// TIA Portal V17 export
// export: Created 2025-05-06T13:48:20.4992801Z, ExportSetting WithDefaults, DisplayName Totally Integrated Automation Portal, DisplayVersion V17 Update 8, DisplayName TIA Portal Openness, DisplayVersion V17 Update 8, DisplayName TIA Portal Version Control Interface, DisplayVersion V17, DisplayName SINAMICS Startdrive Advanced, DisplayVersion V17 SP2, DisplayName SINAMICS Startdrive G110M, G120, G120C, G120D, G120P, G115D, DisplayVersion V17 SP2, DisplayName SINAMICS Startdrive G130, G150, S120, S150, SINAMICS MV, S210, DisplayVersion V17 SP2, DisplayName STEP 7 Professional, DisplayVersion V17 Update 8, DisplayName SINUMERIK ONE STEP 7 Toolbox, DisplayVersion V17 Update 12, DisplayName SINUMERIK 840D sl STEP 7 Toolbox, DisplayVersion V17 Update 12, DisplayName STEP 7 Safety, DisplayVersion V17 Update 6, DisplayName WinCC Advanced, DisplayVersion V17 Update 8
FUNCTION_BLOCK "FB2107_LIGHTS"   // FB2107, LAD
{ S7_Optimized_Access := 'TRUE' }
VERSION : 0.1
// stored: AutoNumber false, IsIECCheckEnabled false, IsRetainMemResEnabled false, MemoryReserve 100, SetENOAutomatically false, UDAEnableTagReadback false
   VAR_INPUT
      GENERAL_MACHINE_LIGHT_OPTION : Bool;
      CIRCUIT_BRAKER_IN : Bool;
      LIGHT_ON_SELECTOR : Bool;
      MANUAL_REQ_LINE : Bool;   // MANUAL REQUEST HMI LINE NUMBER
      SWITCH_ON_AUTO_REQ : Bool;   // SWITCH ON AUTO REQUEST
      SWITCH_OFF_AUTO_REQ : Bool;   // SWITCH OFF AUTO REQUEST
   END_VAR
   VAR_OUTPUT
      LIGHTS_ON : Bool;   // LIGHTS ON OUTPUT
      HMI_LINE_ON_EXEC : Bool;   // HMI LINE ON EXECUTABILITY
      HMI_LINE_OFF_EXEC : Bool;   // HMI LINE OFF EXECUTABILITY
      HMI_LINE_ON_STATUS : Bool;   // HMI LINE ON STATUS
      HMI_LINE_OFF_STATUS : Bool;   // HMI LINE OFF STATUS
   END_VAR
   VAR
      SWITCH_ON_GENERAL_CONDITIONS : Bool;   // SWITCH ON GENERAL CONDITIONS
      SWITCH_ON_INITIAL_CONDITIONS : Bool;   // SWITCH ON INITIAL CONDITIONS
      SWITCH_ON_MANUAL_REQ : Bool;   // SWITCH ON MANUAL REQUEST
      SWITCH_ON_GLOBAL_REQ : Bool;   // SWITCH ON GLOBAL REQUEST
      SWITCH_ON_COMMAND : Bool;   // SWITCH ON COMMAND
      SWITCH_ON : Bool;   // SWITCH ON
      IN_SERVICE : Bool;   // IN SERVICE
      SWITCH_OFF_GENERAL_CONDITIONS : Bool;   // SWITCH OFF GENERAL CONDITIONS
      SWITCH_OFF_INITIAL_CONDITIONS : Bool;   // SWITCH OFF INITIAL CONDITIONS
      SWITCH_OFF_MANUAL_REQ : Bool;   // SWITCH OFF MANUAL REQUEST
      SWITCH_OFF_GLOBAL_REQ : Bool;   // SWITCH OFF GLOBAL REQUEST
      SWITCH_OFF_COMMAND : Bool;   // SWITCH OFF COMMAND
      SWITCH_OFF : Bool;   // SWITCH OFF
      OUT_OF_SERVICE : Bool;   // OUT OF SERVICE
      SWITCH_ON_GLOBAL_REQUEST_AUX0 : Bool;   // SWITCH ON GLOBAL REQUEST AUXILIARY 0
      SWITCH_ON_GLOBAL_REQUEST_AUX1 : Bool;   // SWITCH ON GLOBAL REQUEST AUXILIARY 1
      SWITCH_ON_GLOBAL_REQUEST_AUX2 : Bool;   // SWITCH ON GLOBAL REQUEST AUXILIARY 2
      SWITCH_ON_GLOBAL_REQUEST_AUX3 : Bool;   // SWITCH ON GLOBAL REQUEST AUXILIARY 3
      SWITCH_OFF_GLOBAL_REQUEST_AUX1 : Bool;   // SWITCH OFF GLOBAL REQUEST AUXILIARY 1
      SWITCH_OFF_GLOBAL_REQUEST_AUX2 : Bool;   // SWITCH OFF GLOBAL REQUEST AUXILIARY 2
      SWITCH_OFF_DOORS_CLOSED_TIMER : IEC_TIMER;
      SWITCH_OFF_IN_SERVICE_DELAY_TIMER : IEC_TIMER;
   END_VAR
   // SWITCH_OFF_DOORS_CLOSED_TIMER.PT := T#10M;
   // SWITCH_OFF_IN_SERVICE_DELAY_TIMER.PT := T#1H;
   VAR_TEMP   // added for the SCL form of the ladder/FBD networks
      _w1 : Bool;
      _w2 : Bool;
      _w3 : Bool;
      _w4 : Bool;
      _w5 : Bool;
      _w6 : Bool;
   END_VAR
BEGIN

REGION Network 1: SWITCH ON GENERAL CONDITIONS
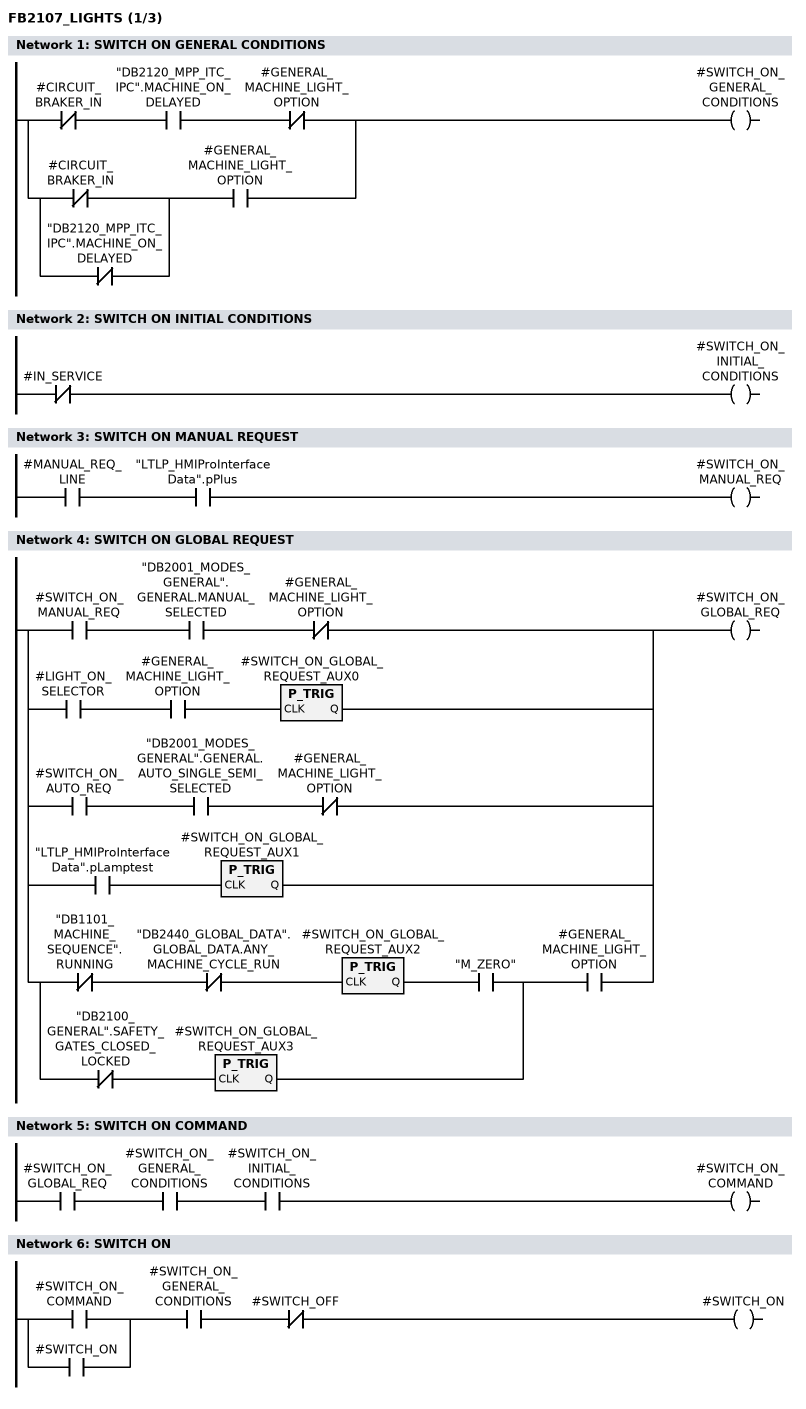
   RUNG wire#powerrail
      I_Contact( #CIRCUIT_BRAKER_IN )
      Contact( "DB2120_MPP_ITC_IPC".MACHINE_ON_DELAYED )
      I_Contact( #GENERAL_MACHINE_LIGHT_OPTION )
      wire#w1
      Coil( #SWITCH_ON_GENERAL_CONDITIONS )
   END_RUNG
   RUNG wire#powerrail
      I_Contact( #CIRCUIT_BRAKER_IN )
      wire#w2
      Contact( #GENERAL_MACHINE_LIGHT_OPTION )
   END_RUNG wire#w1
   RUNG wire#powerrail
      I_Contact( "DB2120_MPP_ITC_IPC".MACHINE_ON_DELAYED )
   END_RUNG wire#w2
   // the same network as SCL:
   #SWITCH_ON_GENERAL_CONDITIONS := (NOT #CIRCUIT_BRAKER_IN AND "DB2120_MPP_ITC_IPC".MACHINE_ON_DELAYED AND NOT #GENERAL_MACHINE_LIGHT_OPTION) OR ((NOT #CIRCUIT_BRAKER_IN OR NOT "DB2120_MPP_ITC_IPC".MACHINE_ON_DELAYED) AND #GENERAL_MACHINE_LIGHT_OPTION);
END_REGION

REGION Network 2: SWITCH ON INITIAL CONDITIONS
   RUNG wire#powerrail
      I_Contact( #IN_SERVICE )
      Coil( #SWITCH_ON_INITIAL_CONDITIONS )
   END_RUNG
   // the same network as SCL:
   #SWITCH_ON_INITIAL_CONDITIONS := NOT #IN_SERVICE;
END_REGION

REGION Network 3: SWITCH ON MANUAL REQUEST
   RUNG wire#powerrail
      Contact( #MANUAL_REQ_LINE )
      Contact( "LTLP_HMIProInterfaceData".pPlus )
      Coil( #SWITCH_ON_MANUAL_REQ )
   END_RUNG
   // the same network as SCL:
   #SWITCH_ON_MANUAL_REQ := #MANUAL_REQ_LINE AND "LTLP_HMIProInterfaceData".pPlus;
END_REGION

REGION Network 4: SWITCH ON GLOBAL REQUEST
   RUNG wire#powerrail
      Contact( #SWITCH_ON_MANUAL_REQ )
      Contact( "DB2001_MODES_GENERAL".GENERAL.MANUAL_SELECTED )
      I_Contact( #GENERAL_MACHINE_LIGHT_OPTION )
      wire#w1
      Coil( #SWITCH_ON_GLOBAL_REQ )
   END_RUNG
   RUNG wire#powerrail
      Contact( #LIGHT_ON_SELECTOR )
      Contact( #GENERAL_MACHINE_LIGHT_OPTION )
      P_Trig( #SWITCH_ON_GLOBAL_REQUEST_AUX0 )
   END_RUNG wire#w1
   RUNG wire#powerrail
      Contact( #SWITCH_ON_AUTO_REQ )
      Contact( "DB2001_MODES_GENERAL".GENERAL.AUTO_SINGLE_SEMI_SELECTED )
      I_Contact( #GENERAL_MACHINE_LIGHT_OPTION )
   END_RUNG wire#w1
   RUNG wire#powerrail
      Contact( "LTLP_HMIProInterfaceData".pLamptest )
      P_Trig( #SWITCH_ON_GLOBAL_REQUEST_AUX1 )
   END_RUNG wire#w1
   RUNG wire#powerrail
      I_Contact( "DB1101_MACHINE_SEQUENCE".RUNNING )
      I_Contact( "DB2440_GLOBAL_DATA".GLOBAL_DATA.ANY_MACHINE_CYCLE_RUN )
      P_Trig( #SWITCH_ON_GLOBAL_REQUEST_AUX2 )
      Contact( "M_ZERO" )
      wire#w2
      Contact( #GENERAL_MACHINE_LIGHT_OPTION )
   END_RUNG wire#w1
   RUNG wire#powerrail
      I_Contact( "DB2100_GENERAL".SAFETY_GATES_CLOSED_LOCKED )
      P_Trig( #SWITCH_ON_GLOBAL_REQUEST_AUX3 )
   END_RUNG wire#w2
   // the same network as SCL:
   #_w1 := #LIGHT_ON_SELECTOR AND #GENERAL_MACHINE_LIGHT_OPTION;
   #_w2 := #_w1 AND NOT #SWITCH_ON_GLOBAL_REQUEST_AUX0;   // rising edge
   #SWITCH_ON_GLOBAL_REQUEST_AUX0 := #_w1;
   #_w3 := "LTLP_HMIProInterfaceData".pLamptest AND NOT #SWITCH_ON_GLOBAL_REQUEST_AUX1;   // rising edge
   #SWITCH_ON_GLOBAL_REQUEST_AUX1 := "LTLP_HMIProInterfaceData".pLamptest;
   #_w4 := NOT "DB1101_MACHINE_SEQUENCE".RUNNING AND NOT "DB2440_GLOBAL_DATA".GLOBAL_DATA.ANY_MACHINE_CYCLE_RUN;
   #_w5 := #_w4 AND NOT #SWITCH_ON_GLOBAL_REQUEST_AUX2;   // rising edge
   #SWITCH_ON_GLOBAL_REQUEST_AUX2 := #_w4;
   #_w6 := NOT "DB2100_GENERAL".SAFETY_GATES_CLOSED_LOCKED AND NOT #SWITCH_ON_GLOBAL_REQUEST_AUX3;   // rising edge
   #SWITCH_ON_GLOBAL_REQUEST_AUX3 := NOT "DB2100_GENERAL".SAFETY_GATES_CLOSED_LOCKED;
   #SWITCH_ON_GLOBAL_REQ := (#SWITCH_ON_MANUAL_REQ AND "DB2001_MODES_GENERAL".GENERAL.MANUAL_SELECTED AND NOT #GENERAL_MACHINE_LIGHT_OPTION) OR #_w2 OR (#SWITCH_ON_AUTO_REQ AND "DB2001_MODES_GENERAL".GENERAL.AUTO_SINGLE_SEMI_SELECTED AND NOT #GENERAL_MACHINE_LIGHT_OPTION) OR #_w3 OR (((#_w5 AND "M_ZERO") OR #_w6) AND #GENERAL_MACHINE_LIGHT_OPTION);
END_REGION

REGION Network 5: SWITCH ON COMMAND
   RUNG wire#powerrail
      Contact( #SWITCH_ON_GLOBAL_REQ )
      Contact( #SWITCH_ON_GENERAL_CONDITIONS )
      Contact( #SWITCH_ON_INITIAL_CONDITIONS )
      Coil( #SWITCH_ON_COMMAND )
   END_RUNG
   // the same network as SCL:
   #SWITCH_ON_COMMAND := #SWITCH_ON_GLOBAL_REQ AND #SWITCH_ON_GENERAL_CONDITIONS AND #SWITCH_ON_INITIAL_CONDITIONS;
END_REGION

REGION Network 6: SWITCH ON
   RUNG wire#powerrail
      Contact( #SWITCH_ON_COMMAND )
      wire#w1
      Contact( #SWITCH_ON_GENERAL_CONDITIONS )
      I_Contact( #SWITCH_OFF )
      Coil( #SWITCH_ON )
   END_RUNG
   RUNG wire#powerrail
      Contact( #SWITCH_ON )
   END_RUNG wire#w1
   // the same network as SCL:
   #SWITCH_ON := (#SWITCH_ON_COMMAND OR #SWITCH_ON) AND #SWITCH_ON_GENERAL_CONDITIONS AND NOT #SWITCH_OFF;
END_REGION

REGION Network 7: IN SERVICE
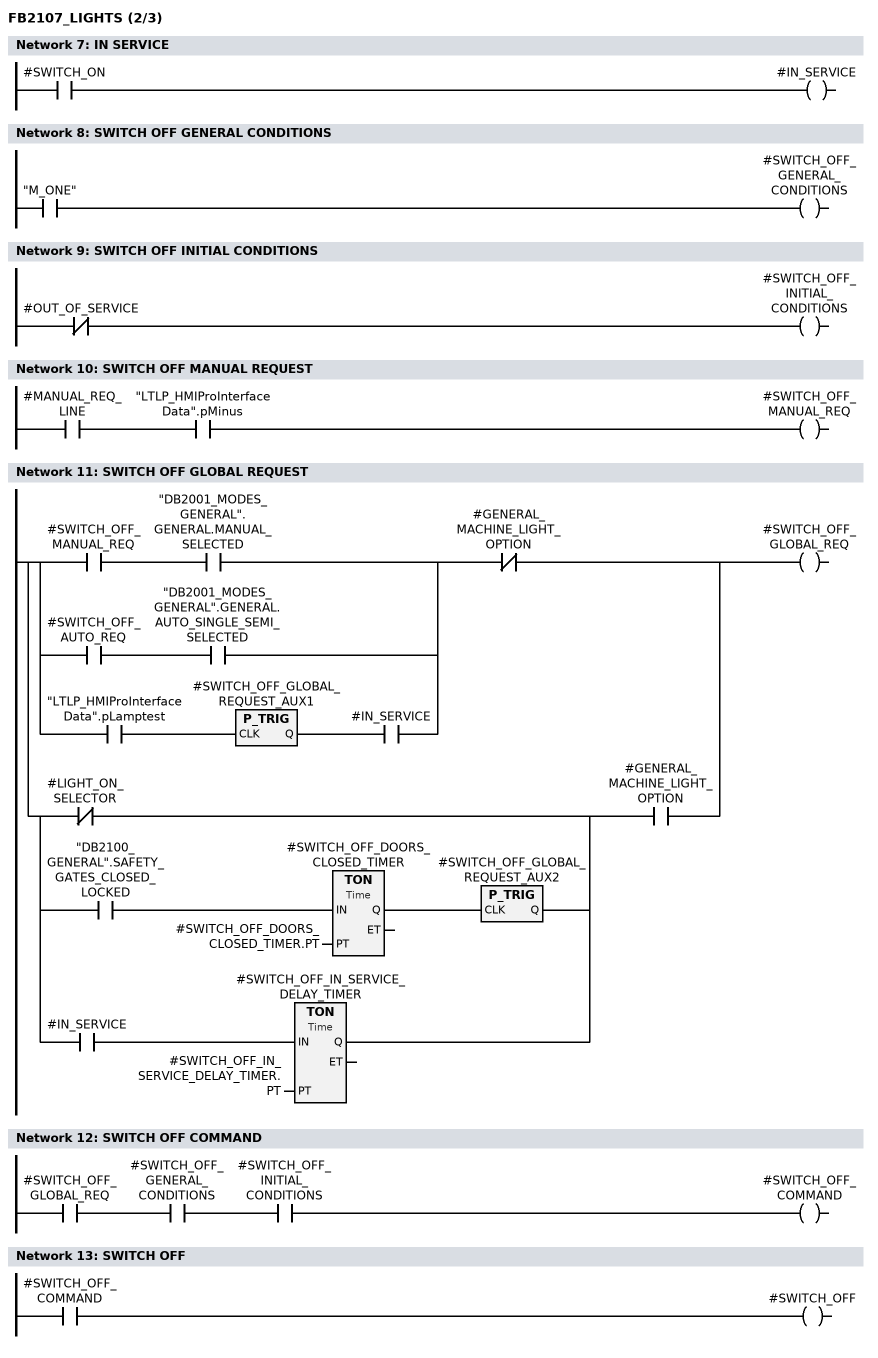
   RUNG wire#powerrail
      Contact( #SWITCH_ON )
      Coil( #IN_SERVICE )
   END_RUNG
   // the same network as SCL:
   #IN_SERVICE := #SWITCH_ON;
END_REGION

REGION Network 8: SWITCH OFF GENERAL CONDITIONS
   RUNG wire#powerrail
      Contact( "M_ONE" )
      Coil( #SWITCH_OFF_GENERAL_CONDITIONS )
   END_RUNG
   // the same network as SCL:
   #SWITCH_OFF_GENERAL_CONDITIONS := "M_ONE";
END_REGION

REGION Network 9: SWITCH OFF INITIAL CONDITIONS
   RUNG wire#powerrail
      I_Contact( #OUT_OF_SERVICE )
      Coil( #SWITCH_OFF_INITIAL_CONDITIONS )
   END_RUNG
   // the same network as SCL:
   #SWITCH_OFF_INITIAL_CONDITIONS := NOT #OUT_OF_SERVICE;
END_REGION

REGION Network 10: SWITCH OFF MANUAL REQUEST
   RUNG wire#powerrail
      Contact( #MANUAL_REQ_LINE )
      Contact( "LTLP_HMIProInterfaceData".pMinus )
      Coil( #SWITCH_OFF_MANUAL_REQ )
   END_RUNG
   // the same network as SCL:
   #SWITCH_OFF_MANUAL_REQ := #MANUAL_REQ_LINE AND "LTLP_HMIProInterfaceData".pMinus;
END_REGION

REGION Network 11: SWITCH OFF GLOBAL REQUEST
   RUNG wire#powerrail
      Contact( #SWITCH_OFF_MANUAL_REQ )
      Contact( "DB2001_MODES_GENERAL".GENERAL.MANUAL_SELECTED )
      wire#w1
      I_Contact( #GENERAL_MACHINE_LIGHT_OPTION )
      wire#w2
      Coil( #SWITCH_OFF_GLOBAL_REQ )
   END_RUNG
   RUNG wire#powerrail
      Contact( #SWITCH_OFF_AUTO_REQ )
      Contact( "DB2001_MODES_GENERAL".GENERAL.AUTO_SINGLE_SEMI_SELECTED )
   END_RUNG wire#w1
   RUNG wire#powerrail
      Contact( "LTLP_HMIProInterfaceData".pLamptest )
      P_Trig( #SWITCH_OFF_GLOBAL_REQUEST_AUX1 )
      Contact( #IN_SERVICE )
   END_RUNG wire#w1
   RUNG wire#powerrail
      I_Contact( #LIGHT_ON_SELECTOR )
      wire#w3
      Contact( #GENERAL_MACHINE_LIGHT_OPTION )
   END_RUNG wire#w2
   RUNG wire#powerrail
      Contact( "DB2100_GENERAL".SAFETY_GATES_CLOSED_LOCKED )
      { S7_Templates := "time_type := Time" } #SWITCH_OFF_DOORS_CLOSED_TIMER.TON(pt := #SWITCH_OFF_DOORS_CLOSED_TIMER.PT, et =>)
      P_Trig( #SWITCH_OFF_GLOBAL_REQUEST_AUX2 )
   END_RUNG wire#w3
   RUNG wire#powerrail
      Contact( #IN_SERVICE )
      { S7_Templates := "time_type := Time" } #SWITCH_OFF_IN_SERVICE_DELAY_TIMER.TON(pt := #SWITCH_OFF_IN_SERVICE_DELAY_TIMER.PT, et =>)
   END_RUNG wire#w3
   // the same network as SCL:
   #_w1 := "LTLP_HMIProInterfaceData".pLamptest AND NOT #SWITCH_OFF_GLOBAL_REQUEST_AUX1;   // rising edge
   #SWITCH_OFF_GLOBAL_REQUEST_AUX1 := "LTLP_HMIProInterfaceData".pLamptest;
   #SWITCH_OFF_DOORS_CLOSED_TIMER.TON(IN := "DB2100_GENERAL".SAFETY_GATES_CLOSED_LOCKED,
                           PT := #SWITCH_OFF_DOORS_CLOSED_TIMER.PT);
   #_w2 := #SWITCH_OFF_DOORS_CLOSED_TIMER.Q AND NOT #SWITCH_OFF_GLOBAL_REQUEST_AUX2;   // rising edge
   #SWITCH_OFF_GLOBAL_REQUEST_AUX2 := #SWITCH_OFF_DOORS_CLOSED_TIMER.Q;
   #SWITCH_OFF_IN_SERVICE_DELAY_TIMER.TON(IN := #IN_SERVICE, PT := #SWITCH_OFF_IN_SERVICE_DELAY_TIMER.PT);
   #SWITCH_OFF_GLOBAL_REQ := (((#SWITCH_OFF_MANUAL_REQ AND "DB2001_MODES_GENERAL".GENERAL.MANUAL_SELECTED) OR (#SWITCH_OFF_AUTO_REQ AND "DB2001_MODES_GENERAL".GENERAL.AUTO_SINGLE_SEMI_SELECTED) OR (#_w1 AND #IN_SERVICE)) AND NOT #GENERAL_MACHINE_LIGHT_OPTION) OR ((NOT #LIGHT_ON_SELECTOR OR #_w2 OR #SWITCH_OFF_IN_SERVICE_DELAY_TIMER.Q) AND #GENERAL_MACHINE_LIGHT_OPTION);
END_REGION

REGION Network 12: SWITCH OFF COMMAND
   RUNG wire#powerrail
      Contact( #SWITCH_OFF_GLOBAL_REQ )
      Contact( #SWITCH_OFF_GENERAL_CONDITIONS )
      Contact( #SWITCH_OFF_INITIAL_CONDITIONS )
      Coil( #SWITCH_OFF_COMMAND )
   END_RUNG
   // the same network as SCL:
   #SWITCH_OFF_COMMAND := #SWITCH_OFF_GLOBAL_REQ AND #SWITCH_OFF_GENERAL_CONDITIONS AND #SWITCH_OFF_INITIAL_CONDITIONS;
END_REGION

REGION Network 13: SWITCH OFF
   RUNG wire#powerrail
      Contact( #SWITCH_OFF_COMMAND )
      Coil( #SWITCH_OFF )
   END_RUNG
   // the same network as SCL:
   #SWITCH_OFF := #SWITCH_OFF_COMMAND;
END_REGION

REGION Network 14: OUT OF SERVICE
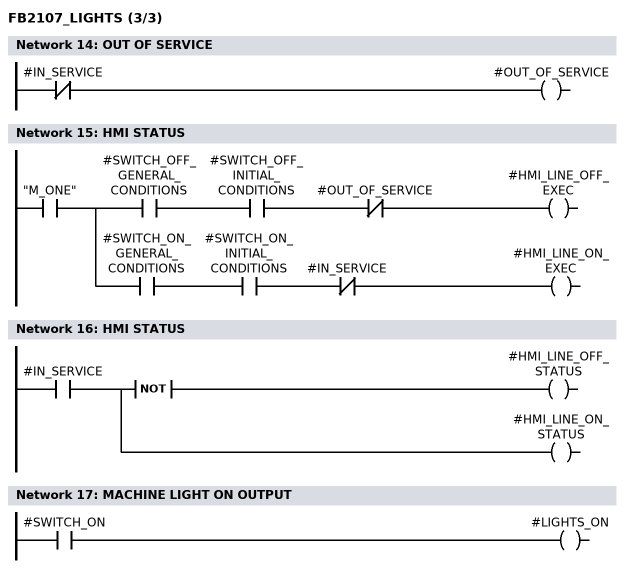
   RUNG wire#powerrail
      I_Contact( #IN_SERVICE )
      Coil( #OUT_OF_SERVICE )
   END_RUNG
   // the same network as SCL:
   #OUT_OF_SERVICE := NOT #IN_SERVICE;
END_REGION

REGION Network 15: HMI STATUS
   RUNG wire#powerrail
      Contact( "M_ONE" )
      wire#w1
      Contact( #SWITCH_OFF_GENERAL_CONDITIONS )
      Contact( #SWITCH_OFF_INITIAL_CONDITIONS )
      I_Contact( #OUT_OF_SERVICE )
      Coil( #HMI_LINE_OFF_EXEC )
   END_RUNG
   RUNG wire#w1
      Contact( #SWITCH_ON_GENERAL_CONDITIONS )
      Contact( #SWITCH_ON_INITIAL_CONDITIONS )
      I_Contact( #IN_SERVICE )
      Coil( #HMI_LINE_ON_EXEC )
   END_RUNG
   // the same network as SCL:
   #HMI_LINE_OFF_EXEC := "M_ONE" AND #SWITCH_OFF_GENERAL_CONDITIONS AND #SWITCH_OFF_INITIAL_CONDITIONS AND NOT #OUT_OF_SERVICE;
   #HMI_LINE_ON_EXEC := "M_ONE" AND #SWITCH_ON_GENERAL_CONDITIONS AND #SWITCH_ON_INITIAL_CONDITIONS AND NOT #IN_SERVICE;
END_REGION

REGION Network 16: HMI STATUS
   RUNG wire#powerrail
      Contact( #IN_SERVICE )
      wire#w1
      Not()
      Coil( #HMI_LINE_OFF_STATUS )
   END_RUNG
   RUNG wire#w1
      Coil( #HMI_LINE_ON_STATUS )
   END_RUNG
   // the same network as SCL:
   #HMI_LINE_OFF_STATUS := NOT #IN_SERVICE;
   #HMI_LINE_ON_STATUS := #IN_SERVICE;
END_REGION

REGION Network 17: MACHINE LIGHT ON OUTPUT
   RUNG wire#powerrail
      Contact( #SWITCH_ON )
      Coil( #LIGHTS_ON )
   END_RUNG
   // the same network as SCL:
   #LIGHTS_ON := #SWITCH_ON;
END_REGION
END_FUNCTION_BLOCK
